// TwinCAT 3 PLC project testStepper
// ProgramVersion: 3.1.4023.0
// libraries:
//   Tc2_MC2, * (Beckhoff Automation GmbH)
//   Tc2_NC, * (Beckhoff Automation GmbH)
//   Tc2_Standard, * (Beckhoff Automation GmbH)
//   Tc2_System, * (Beckhoff Automation GmbH)
//   Tc3_Module, * (Beckhoff Automation GmbH)
//   VisuDialogs, * (System)
// project tree:
//   GlobalPOUs/ MAIN.TcPOU (not stored)
//   / GlobalTextList.TcGTLO (not stored), PlcTask.TcTTO (not stored), Visualization Manager.TcVMO (not stored)
//   GVLs/ GVL_AxisCtr.TcGVL (not stored), GVL_IO.TcGVL, GVL_NC.TcGVL (not stored)
//   Motion_POUs/ Command_to_Action.TcPOU (not stored), DegreesToRelativeMovment.TcPOU (not stored), movements.TcPOU (not stored), PositionToDegree.TcPOU, POUNCPowerOn.TcPOU, Torque_reading.TcPOU (not stored)
//   VISUs/ testStepperVisu.TcVIS (not stored)

// ---- GVLs/GVL_IO.TcGVL
{attribute 'qualified_only'}
VAR_GLOBAL
	I_bXAxisLimitSwPos AT %I* : BOOL;
	I_bXAxisLimitSwNeg AT %I* : BOOL;
	
END_VAR

// ---- Motion_POUs/PositionToDegree.TcPOU
FUNCTION_BLOCK PositionToDegree
VAR_INPUT
	MaxPosition : LREAL;
	MaxSteeringAngle : INT;
	Position : LREAL;
END_VAR
VAR_OUTPUT
	Deg : LREAL;
END_VAR
VAR
END_VAR

IF (Position > 0 OR Position < 0) THEN
	Deg := (MaxSteeringAngle/MaxPosition)*Position;
ELSIF (Position = 0) THEN
	Deg := 0;		
END_IF

END_FUNCTION_BLOCK

// ---- Motion_POUs/POUNCPowerOn.TcPOU
PROGRAM POUNCPowerOn
VAR
	fbXAxisPowerOn : MC_Power;
	fbXAxisDrive : MC_MoveRelative;
	DegreesToRelativeMovment_0: DegreesToRelativeMovment;
	HomingActive: BOOL;
	MC_Home_0: MC_Home;
	StartHoming: BOOL;
	endSW: BOOL;
	MC_Reset_0: MC_Reset;
	reset: BOOL;
	
	
	//command : STRING;
END_VAR

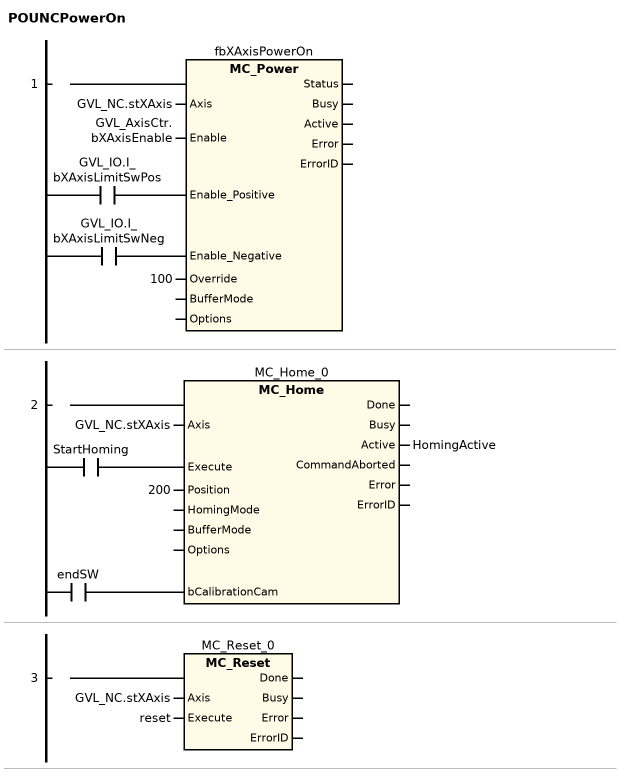
// NETWORK 1
fbXAxisPowerOn(
    Axis := GVL_NC.stXAxis,
    Enable := GVL_AxisCtr.bXAxisEnable,
    Enable_Positive := GVL_IO.I_bXAxisLimitSwPos,
    Enable_Negative := GVL_IO.I_bXAxisLimitSwNeg,
    Override := 100); // MC_Power

// NETWORK 2
MC_Home_0(
    Axis := GVL_NC.stXAxis,
    Execute := StartHoming,
    Position := 200,
    bCalibrationCam := endSW,
    Active => HomingActive); // MC_Home

// NETWORK 3
MC_Reset_0(Axis := GVL_NC.stXAxis, Execute := reset); // MC_Reset

END_PROGRAM
